FUNCTION_BLOCK FB_FT_PD (* Composite Function Block Type *)
  (* Standard: 61499-2 *)
  (* Version 0.0, 2011-08-27, 4DIAC-IDE, 4DIAC-Consortium *)
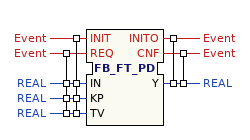
  EVENT_INPUT
    INIT WITH IN, KP, TV; (* Initialization Request *)
    REQ WITH IN, KP, TV; (* Normal Execution Request *)
  END_EVENT
  EVENT_OUTPUT
    INITO WITH Y; (* Initialization Confirm *)
    CNF WITH Y; (* Execution Confirmation *)
  END_EVENT
  VAR_INPUT
    IN : REAL; (* input signal *)
    KP : REAL := 1.0; (* proportional part of the controller *)
    TV : REAL := 1.0; (* reset time of the differentiator in seconds *)
  END_VAR
  VAR_OUTPUT
    Y : REAL; (* Output event qualifier *)
  END_VAR
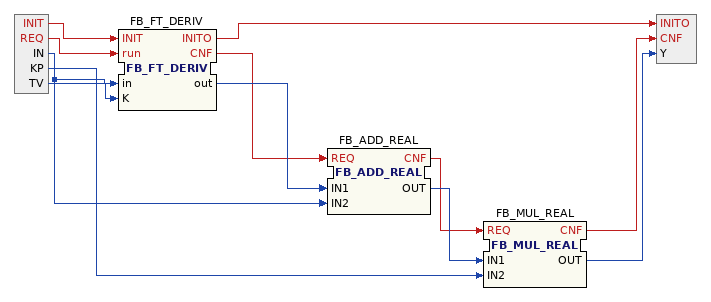
  FBS
    FB_FT_DERIV : FB_FT_DERIV;
    FB_ADD_REAL : FB_ADD_REAL;
    FB_MUL_REAL : FB_MUL_REAL;
  END_FBS
  EVENT_CONNECTIONS
    INIT TO FB_FT_DERIV.INIT;
    FB_FT_DERIV.INITO TO INITO;
    REQ TO FB_FT_DERIV.run;
    FB_FT_DERIV.CNF TO FB_ADD_REAL.REQ;
    FB_ADD_REAL.CNF TO FB_MUL_REAL.REQ;
    FB_MUL_REAL.CNF TO CNF;
  END_CONNECTIONS
  DATA_CONNECTIONS
    TV TO FB_FT_DERIV.K;
    IN TO FB_FT_DERIV.in;
    FB_FT_DERIV.out TO FB_ADD_REAL.IN1;
    IN TO FB_ADD_REAL.IN2;
    FB_ADD_REAL.OUT TO FB_MUL_REAL.IN1;
    KP TO FB_MUL_REAL.IN2;
    FB_MUL_REAL.OUT TO Y;
  END_CONNECTIONS
END_FUNCTION_BLOCK
